INTERFACE IPluginRunner EXTENDS __System.IQueryInterface

METHOD RegisterPlugin
VAR_INPUT
	plugin : IPlugin;
END_VAR
END_METHOD

END_INTERFACE

(* stored: Version 1.1.0.1, ProductVersion 3.1.4024.12
   Itf IPluginRunner: Id {81c261ba-8c6e-4e80-a41e-8f5e19ff3c9a}
   Method RegisterPlugin: Id {b3d01674-ef9b-472d-9fde-029420df9f2f} *)
